FUNCTION_BLOCK FBlock (* Basic function block *)
  (* Standard: 61499 *)
  (* Version 1.0, 11/20/2015 9:00 AM, Kawsihen, Kawsihen_s Macintosh *)
  (* Compiler header: package mypackage *)
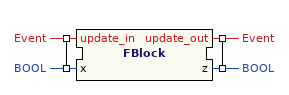
  EVENT_INPUT
    update_in WITH x;
  END_EVENT
  EVENT_OUTPUT
    update_out WITH z;
  END_EVENT
  VAR_INPUT
    x : BOOL;
  END_VAR
  VAR_OUTPUT
    z : BOOL;
  END_VAR
  VAR
    k : REAL;
    d : REAL;
    signal : REAL;
    y : REAL;
    C1y : REAL;
  END_VAR
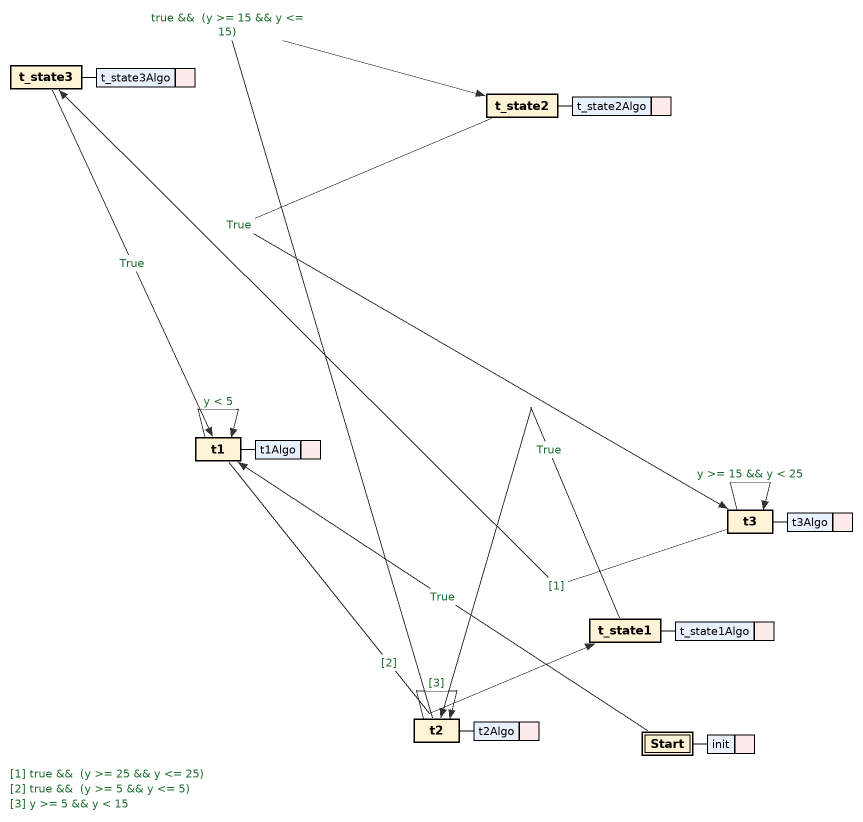
  EC_STATES
    Start : init;
    t1 : t1Algo;
    t2 : t2Algo;
    t3 : t3Algo;
    t_state1 : t_state1Algo;
    t_state2 : t_state2Algo;
    t_state3 : t_state3Algo;
  END_STATES
  EC_TRANSITIONS
    Start TO t1 := True;
    t1 TO t_state1 := true &&  (y >= 5 && y <= 5);
    t_state1 TO t2 := True;
    t2 TO t_state2 := true &&  (y >= 15 && y <= 15);
    t_state2 TO t3 := True;
    t3 TO t_state3 := true &&  (y >= 25 && y <= 25);
    t_state3 TO t1 := True;
    t1 TO t1 := y < 5;
    t2 TO t2 := y >= 5 && y < 15;
    t3 TO t3 := y >= 15 && y < 25;
  END_TRANSITIONS
  ALGORITHM t1Algo IN C:
me->C1y = 0;
me->y = (float) me->C1y + me->d*me->k;
me->k++;
  END_ALGORITHM
  ALGORITHM t2Algo IN C:
me->C1y = 0;
me->y = (float) me->C1y + me->d*me->k;
me->k++;
  END_ALGORITHM
  ALGORITHM t3Algo IN C:
me->C1y = 0;
me->y = (float) me->C1y + me->d*me->k;
me->k++;
  END_ALGORITHM
  ALGORITHM init IN C:
me->d = 0.01;
me->k = 0;
  END_ALGORITHM
  ALGORITHM t_state1Algo IN C:
me->y = me->y;
me->signal = 1;
me->k = 0;
  END_ALGORITHM
  ALGORITHM t_state2Algo IN C:
me->y = me->y;
me->signal = 0;
me->k = 0;
  END_ALGORITHM
  ALGORITHM t_state3Algo IN C:
me->y = 0;
me->k = 0;
  END_ALGORITHM
END_FUNCTION_BLOCK
